FUNCTION_BLOCK FIND_P (* Find the beginning character position of the first occurrence of IN1 in IN2 following position P *)
  (* Standard: 61131-3 *)
  (* Version 0.0, 2004-12-15, JHC, Rockwell Automation, Converted from SRC format. *)
  (* Compiler header: package fb.rt.plc.strings; *)
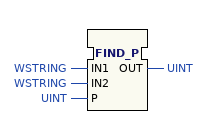
  VAR_INPUT
    IN1 : WSTRING;
    IN2 : WSTRING;
    P : UINT;
  END_VAR
  VAR_OUTPUT
    OUT : UINT;
  END_VAR
END_FUNCTION_BLOCK
